// TIA Portal V18 export
FUNCTION_BLOCK "Cycle_iterator_spot_generator"   // FB78, FBD
{ S7_Optimized_Access := 'TRUE' }
VERSION : 0.1
// stored: AutoNumber true, IsIECCheckEnabled false, IsRetainMemResEnabled false, MemoryReserve 100, SetENOAutomatically false, UDAEnableTagReadback false
   VAR_INPUT
      cur_pos : "typePositions";
      "step" : Real;
      fullturn : Real;
   END_VAR
   VAR_OUTPUT
      list : "typeSpotList";
      ER : Bool;
   END_VAR
   VAR
      j : Int;
   END_VAR
   VAR_TEMP
      N : Real;
   END_VAR
BEGIN

REGION Network 1 (SCL)
   #N := #fullturn / #step;

   #list.N := DINT_TO_INT(CEIL(#N));
END_REGION

REGION Network 2 (SCL)

   #ER := FALSE;

   IF #fullturn > 0.0 AND #step > 0 AND #step < #fullturn AND #list.N > 1 AND #list.N <= "_SPOT_DB".Spot_N_max THEN
       FOR #j := 1 TO #list.N DO
           #list.pos_AR[#j] := #cur_pos;
           #list.pos_AR[#j].M5O2 := #step * INT_TO_REAL(#j - 1);
       END_FOR;

   ELSE
       #ER := true;
   END_IF;
END_REGION
END_FUNCTION_BLOCK
